FUNCTION_BLOCK Composite (* Composite Function Block Type *)
  (* Standard: 61499-2 *)
  (* Version 0.2, 2003-12-05, JHC, Rockwell Automation, Renamed from NEWCOMPFB. *)
  (* Version 0.1, 2002-01-08, JHC, Rockwell Automation, Added DLY FB as example. *)
  (* Version 0.0, 2000-05-27, JHC, Rockwell Automation *)
  (* Compiler header: package fb.rt.cs725; *)
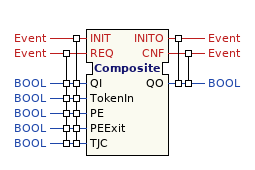
  EVENT_INPUT
    INIT WITH QI, TokenIn, PE, PEExit, TJC; (* Initialization Request *)
    REQ WITH QI, TokenIn, PE, PEExit, TJC; (* Normal Execution Request *)
  END_EVENT
  EVENT_OUTPUT
    INITO WITH QO; (* Initialization Confirm *)
    CNF WITH QO; (* Execution Confirmation *)
  END_EVENT
  VAR_INPUT
    QI : BOOL; (* Input event qualifier *)
    TokenIn : BOOL;
    PE : BOOL;
    PEExit : BOOL;
    TJC : BOOL;
  END_VAR
  VAR_OUTPUT
    QO : BOOL; (* Output event qualifier *)
  END_VAR
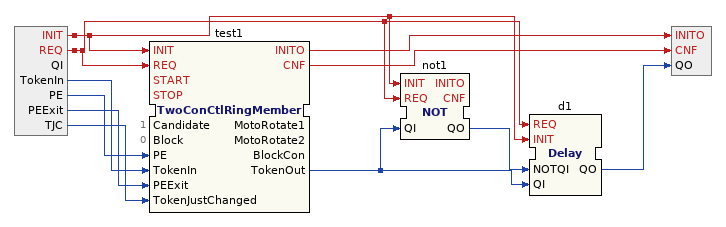
  FBS
    test1 : TwoConCtlRingMember(Candidate := 1, Block := 0);
    not1 : NOT;
    d1 : Delay;
  END_FBS
  EVENT_CONNECTIONS
    REQ TO test1.REQ;
    INIT TO test1.INIT;
    test1.CNF TO CNF;
    test1.INITO TO INITO;
    REQ TO d1.REQ;
    INIT TO d1.INIT;
    INIT TO not1.INIT;
    REQ TO not1.REQ;
  END_CONNECTIONS
  DATA_CONNECTIONS
    test1.TokenOut TO not1.QI;
    not1.QO TO d1.NOTQI;
    test1.TokenOut TO d1.QI;
    d1.QO TO QO;
    PE TO test1.PE;
    TokenIn TO test1.TokenIn;
    PEExit TO test1.PEExit;
    TJC TO test1.TokenJustChanged;
  END_CONNECTIONS
END_FUNCTION_BLOCK
